FUNCTION And4 : BoolValue
VAR_INPUT
	value1 : BoolValue;
	value2 : BoolValue;
	value3 : BoolValue;
	value4 : BoolValue;
END_VAR
VAR
	p : POINTER TO BooleanExpression;
END_VAR

p := __NEW(BooleanExpression);

p^.Op4(
	operator := BooleanOperator.ANDop,
	value1 := value1,
	value2 := value2,
	value3 := value3,
	value4 := value4
);

And4 := p^;

END_FUNCTION

(* stored: Version 1.1.0.1
   POU And4: Id {097e1958-6933-4acc-86cb-af30df9f2525}, SpecialFunc None *)
